FUNCTION_BLOCK FB_System_BHKW_Ablaufsteuerung
VAR_IN_OUT
	Zustand					: ST_System_BHKW_Zustand;
	Stellwert				: ST_System_BHKW_Stellwert;
	Steuerung				: ST_System_BHKW_Steuerung;
	Parameter				: ST_System_BHKW_Parameter;
END_VAR
VAR_INPUT
	Zustand_Stellventil		: ST_SVs_Zustand;
	Zustand_Pumpe			: ST_PU_Zustand;
	Zustand_BHKW			: ST_BHKW_Zustand;
END_VAR
VAR_OUTPUT
END_VAR
VAR
	Timer1					: TON;
	Timer2					: TON;
	Timer3					: TOF;
END_VAR

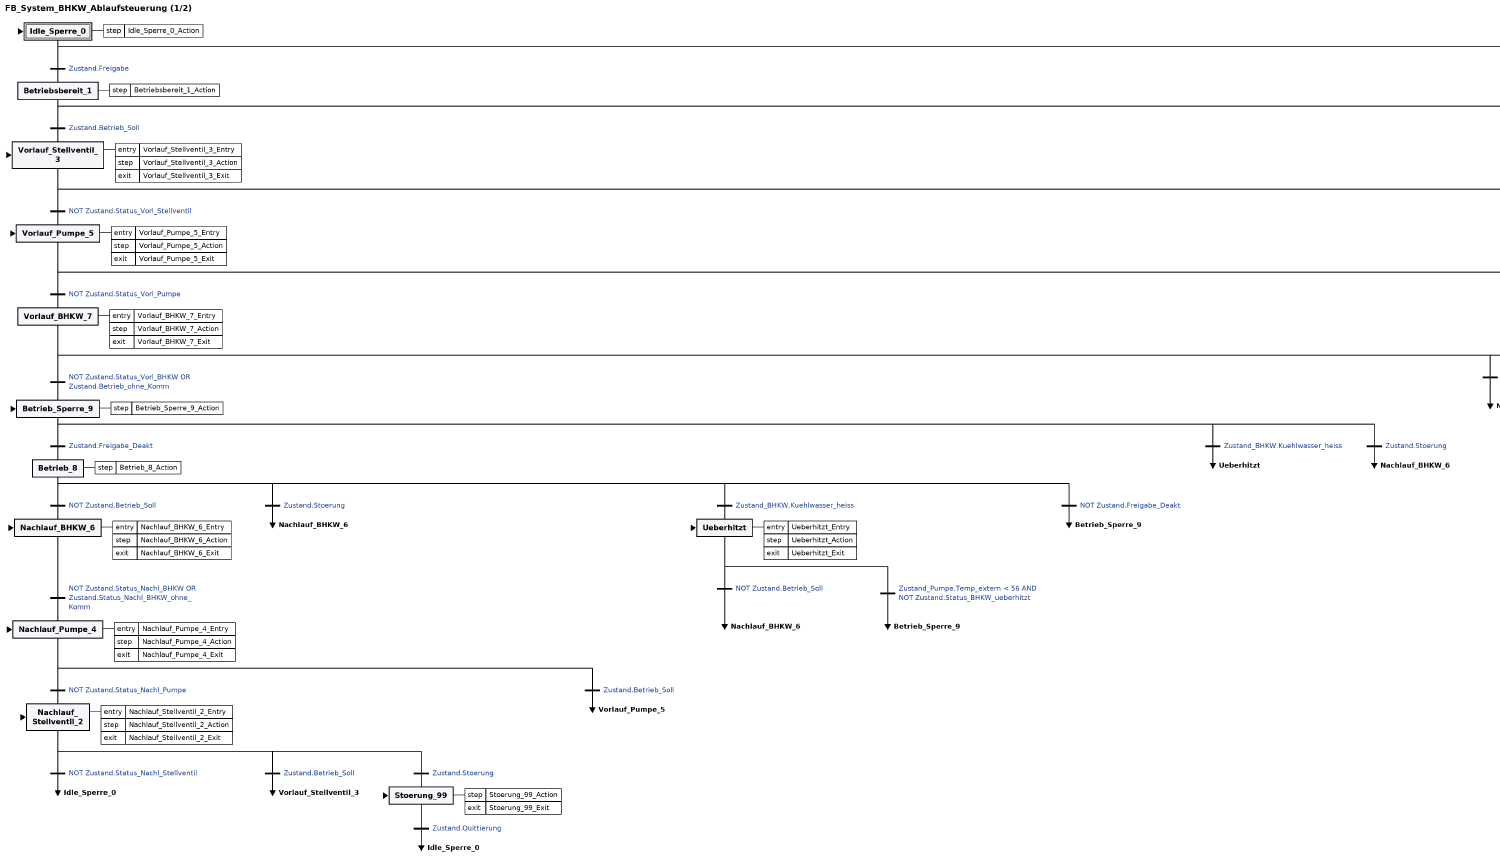
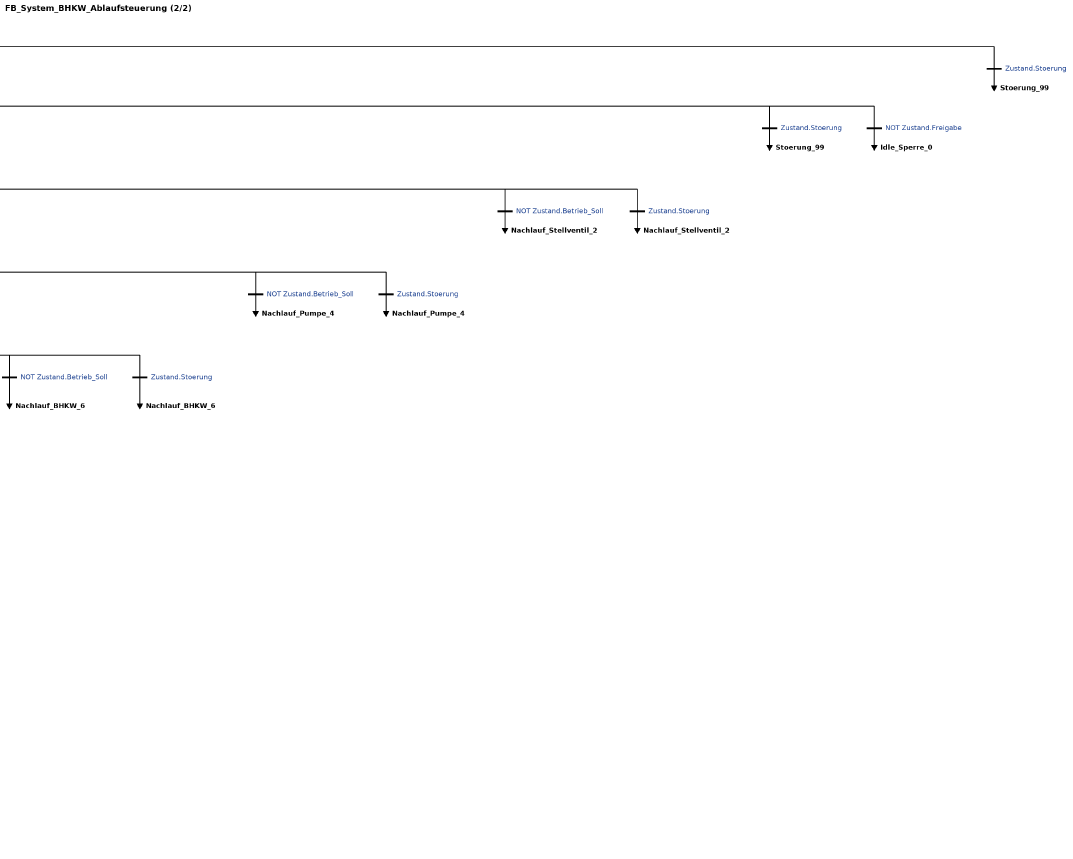
INITIAL_STEP Idle_Sperre_0:
    Idle_Sperre_0_Action(N);  // step action
END_STEP
TRANSITION FROM Idle_Sperre_0 TO Betriebsbereit_1
    := Zustand.Freigabe;
END_TRANSITION
TRANSITION FROM Idle_Sperre_0 TO Stoerung_99
    := Zustand.Stoerung;
END_TRANSITION
STEP Betriebsbereit_1:
    Betriebsbereit_1_Action(N);  // step action
END_STEP
TRANSITION FROM Betriebsbereit_1 TO Vorlauf_Stellventil_3
    := Zustand.Betrieb_Soll;
END_TRANSITION
TRANSITION FROM Betriebsbereit_1 TO Stoerung_99
    := Zustand.Stoerung;
END_TRANSITION
TRANSITION FROM Betriebsbereit_1 TO Idle_Sperre_0
    := NOT Zustand.Freigabe;
END_TRANSITION
STEP Vorlauf_Stellventil_3:
    Vorlauf_Stellventil_3_Entry(P1);  // entry action
    Vorlauf_Stellventil_3_Action(N);  // step action
    Vorlauf_Stellventil_3_Exit(P0);  // exit action
END_STEP
TRANSITION FROM Vorlauf_Stellventil_3 TO Vorlauf_Pumpe_5
    := NOT Zustand.Status_Vorl_Stellventil;
END_TRANSITION
TRANSITION FROM Vorlauf_Stellventil_3 TO Nachlauf_Stellventil_2
    := NOT Zustand.Betrieb_Soll;
END_TRANSITION
TRANSITION FROM Vorlauf_Stellventil_3 TO Nachlauf_Stellventil_2
    := Zustand.Stoerung;
END_TRANSITION
STEP Vorlauf_Pumpe_5:
    Vorlauf_Pumpe_5_Entry(P1);  // entry action
    Vorlauf_Pumpe_5_Action(N);  // step action
    Vorlauf_Pumpe_5_Exit(P0);  // exit action
END_STEP
TRANSITION FROM Vorlauf_Pumpe_5 TO Vorlauf_BHKW_7
    := NOT Zustand.Status_Vorl_Pumpe;
END_TRANSITION
TRANSITION FROM Vorlauf_Pumpe_5 TO Nachlauf_Pumpe_4
    := NOT Zustand.Betrieb_Soll;
END_TRANSITION
TRANSITION FROM Vorlauf_Pumpe_5 TO Nachlauf_Pumpe_4
    := Zustand.Stoerung;
END_TRANSITION
STEP Vorlauf_BHKW_7:
    Vorlauf_BHKW_7_Entry(P1);  // entry action
    Vorlauf_BHKW_7_Action(N);  // step action
    Vorlauf_BHKW_7_Exit(P0);  // exit action
END_STEP
TRANSITION FROM Vorlauf_BHKW_7 TO Betrieb_Sperre_9
    := NOT Zustand.Status_Vorl_BHKW OR Zustand.Betrieb_ohne_Komm;
END_TRANSITION
TRANSITION FROM Vorlauf_BHKW_7 TO Nachlauf_BHKW_6
    := NOT Zustand.Betrieb_Soll;
END_TRANSITION
TRANSITION FROM Vorlauf_BHKW_7 TO Nachlauf_BHKW_6
    := Zustand.Stoerung;
END_TRANSITION
STEP Betrieb_Sperre_9:
    Betrieb_Sperre_9_Action(N);  // step action
END_STEP
TRANSITION FROM Betrieb_Sperre_9 TO Betrieb_8
    := Zustand.Freigabe_Deakt;
END_TRANSITION
TRANSITION FROM Betrieb_Sperre_9 TO Ueberhitzt
    := Zustand_BHKW.Kuehlwasser_heiss;
END_TRANSITION
TRANSITION FROM Betrieb_Sperre_9 TO Nachlauf_BHKW_6
    := Zustand.Stoerung;
END_TRANSITION
STEP Betrieb_8:
    Betrieb_8_Action(N);  // step action
END_STEP
TRANSITION FROM Betrieb_8 TO Nachlauf_BHKW_6
    := NOT Zustand.Betrieb_Soll;
END_TRANSITION
TRANSITION FROM Betrieb_8 TO Nachlauf_BHKW_6
    := Zustand.Stoerung;
END_TRANSITION
TRANSITION FROM Betrieb_8 TO Ueberhitzt
    := Zustand_BHKW.Kuehlwasser_heiss;
END_TRANSITION
STEP Ueberhitzt:
    Ueberhitzt_Entry(P1);  // entry action
    Ueberhitzt_Action(N);  // step action
    Ueberhitzt_Exit(P0);  // exit action
END_STEP
TRANSITION FROM Ueberhitzt TO Nachlauf_BHKW_6
    := NOT Zustand.Betrieb_Soll;
END_TRANSITION
TRANSITION FROM Ueberhitzt TO Betrieb_Sperre_9
    := Zustand_Pumpe.Temp_extern < 56 AND NOT Zustand.Status_BHKW_ueberhitzt;
END_TRANSITION
TRANSITION FROM Betrieb_8 TO Betrieb_Sperre_9
    := NOT Zustand.Freigabe_Deakt;
END_TRANSITION
STEP Nachlauf_BHKW_6:
    Nachlauf_BHKW_6_Entry(P1);  // entry action
    Nachlauf_BHKW_6_Action(N);  // step action
    Nachlauf_BHKW_6_Exit(P0);  // exit action
END_STEP
TRANSITION FROM Nachlauf_BHKW_6 TO Nachlauf_Pumpe_4
    := NOT Zustand.Status_Nachl_BHKW OR Zustand.Status_Nachl_BHKW_ohne_Komm;
END_TRANSITION
STEP Nachlauf_Pumpe_4:
    Nachlauf_Pumpe_4_Entry(P1);  // entry action
    Nachlauf_Pumpe_4_Action(N);  // step action
    Nachlauf_Pumpe_4_Exit(P0);  // exit action
END_STEP
TRANSITION FROM Nachlauf_Pumpe_4 TO Nachlauf_Stellventil_2
    := NOT Zustand.Status_Nachl_Pumpe;
END_TRANSITION
TRANSITION FROM Nachlauf_Pumpe_4 TO Vorlauf_Pumpe_5
    := Zustand.Betrieb_Soll;
END_TRANSITION
STEP Nachlauf_Stellventil_2:
    Nachlauf_Stellventil_2_Entry(P1);  // entry action
    Nachlauf_Stellventil_2_Action(N);  // step action
    Nachlauf_Stellventil_2_Exit(P0);  // exit action
END_STEP
TRANSITION FROM Nachlauf_Stellventil_2 TO Idle_Sperre_0
    := NOT Zustand.Status_Nachl_Stellventil;
END_TRANSITION
TRANSITION FROM Nachlauf_Stellventil_2 TO Vorlauf_Stellventil_3
    := Zustand.Betrieb_Soll;
END_TRANSITION
TRANSITION FROM Nachlauf_Stellventil_2 TO Stoerung_99
    := Zustand.Stoerung;
END_TRANSITION
STEP Stoerung_99:
    Stoerung_99_Action(N);  // step action
    Stoerung_99_Exit(P0);  // exit action
END_STEP
TRANSITION FROM Stoerung_99 TO Idle_Sperre_0
    := Zustand.Quittierung;
END_TRANSITION

ACTION Betrieb_8_Action:
(* Stellwert setzen *)
Stellwert.Anford_Stellventil		:= TRUE;
Stellwert.Anford_Pumpe		:= TRUE;
Stellwert.Anford_BHKW			:= TRUE;

(* Zustand setzen *)
Zustand.Status				:= E_System_BHKW_Zustand_Status_Betrieb;
END_ACTION

ACTION Betrieb_Sperre_9_Action:
(* Stellwert setzen *)
Stellwert.Anford_Stellventil		:= TRUE;
Stellwert.Anford_Pumpe		:= TRUE;
Stellwert.Anford_BHKW			:= TRUE;

(* Zustand setzen *)
Zustand.Status				:= E_System_BHKW_Zustand_Status_Betrieb_Sperre;
END_ACTION

ACTION Betriebsbereit_1_Action:
(* Stellwert setzen *)
Stellwert.Anford_Stellventil	:= FALSE;
Stellwert.Anford_Pumpe	:= FALSE;
Stellwert.Anford_BHKW		:= FALSE;

(* Zustand setzen *)
Zustand.Status			:= E_System_BHKW_Zustand_Status_Betriebsbereit;
END_ACTION

ACTION Idle_Sperre_0_Action:
(* Stellwert setzen *)
Stellwert.Anford_Stellventil	:= FALSE;
Stellwert.Anford_Pumpe	:= FALSE;
Stellwert.Anford_BHKW		:= FALSE;

(* Zustand setzen *)
Zustand.Status			:= E_System_BHKW_Zustand_Status_Idle_Sperre;
Zustand.Betrieb_ohne_Komm	:= FALSE;


(* Quittierungszustand auf False setzen, damit das System bei einer erneuten Störung nicht direkt wieder angeschaltet wird *)
Steuerung.Quittierung	:= FALSE;
END_ACTION

ACTION Nachlauf_BHKW_6_Action:
(* Stellwert setzen *)
Stellwert.Anford_Stellventil		:= TRUE;
Stellwert.Anford_Pumpe		:= TRUE;
Stellwert.Anford_BHKW			:= FALSE;

(* Zustand setzen *)
Zustand.Status				:= E_System_BHKW_Zustand_Status_Nachl_BHKW;
Zustand_BHKW.Status_Nachl;
Zustand.Status_Nachl_BHKW	:= Zustand_BHKW.Betrieb OR Zustand_BHKW.Status_Nachl;


(* falls es keine Rückmeldung vom BHKW-Kommunikationsmodul gibt, geht der Nachlauf dennoch weiter *)
Timer2(	IN := Zustand.Status_Nachl_BHKW,
		PT := Parameter.Zeit_Nachl,
		Q => Zustand.Status_Nachl_BHKW_ohne_Komm
);
Zustand.Status_Nachl_BHKW_ohne_Komm := NOT Zustand.Status_Nachl_BHKW_ohne_Komm;
END_ACTION

ACTION Nachlauf_BHKW_6_Entry:
Zustand.Status_Nachl_BHKW			:= TRUE;
Zustand.Status_Nachl_BHKW_ohne_Komm := TRUE;
END_ACTION

ACTION Nachlauf_BHKW_6_Exit:
Zustand.Status_Nachl_BHKW			:= FALSE;
Zustand.Status_Nachl_BHKW_ohne_Komm := FALSE;
END_ACTION

ACTION Nachlauf_Pumpe_4_Action:
(* Stellwert setzen *)
Stellwert.Anford_Stellventil		:= TRUE;
Stellwert.Anford_Pumpe				:= FALSE;
Stellwert.Anford_BHKW				:= FALSE;

(* Zustand setzen *)
Zustand.Status				:= E_System_BHKW_Zustand_Status_Nachl_Pumpe;
Zustand.Status_Nachl_Pumpe	:= Zustand_Pumpe.Betrieb OR Zustand_Pumpe.Status_Nachl;
END_ACTION

ACTION Nachlauf_Pumpe_4_Entry:
Zustand.Status_Nachl_Pumpe	:= TRUE;
END_ACTION

ACTION Nachlauf_Pumpe_4_Exit:
Zustand.Status_Nachl_Pumpe	:= FALSE;
END_ACTION

ACTION Nachlauf_Stellventil_2_Action:
(* Stellwert setzen *)
Stellwert.Anford_Stellventil		:= FALSE;
Stellwert.Anford_Pumpe		:= FALSE;
Stellwert.Anford_BHKW			:= FALSE;

(* Zustand setzen *)
Zustand.Status				:= E_System_BHKW_Zustand_Status_Nachl_Stellventil;
Zustand.Status_Nachl_Stellventil	:= Zustand_Stellventil.Stellung OR Zustand_Stellventil.Stellungwechsel10;
END_ACTION

ACTION Nachlauf_Stellventil_2_Entry:
Zustand.Status_Nachl_Stellventil	:= TRUE;
END_ACTION

ACTION Nachlauf_Stellventil_2_Exit:
Zustand.Status_Nachl_Stellventil	:= FALSE;
END_ACTION

ACTION Stoerung_99_Action:
(* Stellwert setzen *)
Stellwert.Anford_Stellventil	:= FALSE;
Stellwert.Anford_Pumpe	:= FALSE;
Stellwert.Anford_BHKW		:= FALSE;

(* Zustand setzen *)
Zustand.Stoerung			:= TRUE;
Zustand.Status			:= E_System_BHKW_Zustand_Status_Stoerung;
END_ACTION

ACTION Stoerung_99_Exit:
Zustand.Stoerung	:= FALSE;
END_ACTION

ACTION Ueberhitzt_Action:
(* Stellwert setzen *)
Stellwert.Anford_Stellventil	:= TRUE;
Stellwert.Anford_Pumpe			:= TRUE;
Stellwert.Anford_BHKW			:= FALSE;

(* Zustand setzen *)
Zustand.Status				:= E_System_BHKW_Zustand_Status_Ueberhitzt;

(* Mindestens eine halbe Stunde abkühlen *)
Timer3( IN := Zustand_BHKW.Kuehlwasser_heiss,
		PT := T#30M
);

Zustand.Status_BHKW_ueberhitzt := Timer3.Q;
END_ACTION

ACTION Ueberhitzt_Entry:
Zustand.Status_BHKW_ueberhitzt := TRUE;
(* Reset Timer *)
Timer3(IN := FALSE);
END_ACTION

ACTION Ueberhitzt_Exit:
Zustand.Status_BHKW_ueberhitzt := FALSE;
(* Reset Timer *)
Timer3(IN := FALSE);
END_ACTION

ACTION Vorlauf_BHKW_7_Action:
(* Stellwert setzen *)
Stellwert.Anford_Stellventil		:= TRUE;
Stellwert.Anford_Pumpe		:= TRUE;
Stellwert.Anford_BHKW			:= TRUE;

(* Zustand setzen *)
Zustand.Status				:= E_System_BHKW_Zustand_Status_Vorl_BHKW;
Zustand.Status_Vorl_BHKW		:= NOT(Zustand_BHKW.Betrieb AND NOT Zustand_BHKW.Status_Vorl);


(* falls keine Rückmeldung vom BHKW-Kommunikationsmodul kommt, wird der Zustand dennoch auf Betrieb gesetzt *)
Timer1(	IN := Zustand.Status_Vorl_BHKW,
		PT := Parameter.Zeit_Vorl,
		Q => Zustand.Betrieb_ohne_Komm
);
END_ACTION

ACTION Vorlauf_BHKW_7_Entry:
Zustand.Status_Vorl_BHKW		:= TRUE;
END_ACTION

ACTION Vorlauf_BHKW_7_Exit:
Zustand.Status_Vorl_BHKW		:= FALSE;
END_ACTION

ACTION Vorlauf_Pumpe_5_Action:
(* Stellwert setzen *)
Stellwert.Anford_Stellventil		:= TRUE;
Stellwert.Anford_Pumpe		:= TRUE;
Stellwert.Anford_BHKW			:= FALSE;

(* Zustand setzen *)
Zustand.Status				:= E_System_BHKW_Zustand_Status_Vorl_Pumpe;
Zustand.Status_Vorl_Pumpe	:= NOT(Zustand_Pumpe.Betrieb AND NOT Zustand_Pumpe.Status_Vorl);
END_ACTION

ACTION Vorlauf_Pumpe_5_Entry:
Zustand.Status_Vorl_Pumpe	:= TRUE;
END_ACTION

ACTION Vorlauf_Pumpe_5_Exit:
Zustand.Status_Vorl_Pumpe	:= FALSE;
END_ACTION

ACTION Vorlauf_Stellventil_3_Action:
(* Stellwert setzen *)
Stellwert.Anford_Stellventil		:= TRUE;
Stellwert.Anford_Pumpe		:= FALSE;
Stellwert.Anford_BHKW			:= FALSE;

(* Zustand setzen *)
Zustand.Status				:= E_System_BHKW_Zustand_Status_Vorl_Stellventil;
Zustand.Status_Vorl_Stellventil	:= NOT(Zustand_Stellventil.Stellung AND NOT Zustand_Stellventil.Stellungwechsel01);
END_ACTION

ACTION Vorlauf_Stellventil_3_Entry:
Zustand.Status_Vorl_Stellventil	:= TRUE;
END_ACTION

ACTION Vorlauf_Stellventil_3_Exit:
Zustand.Status_Vorl_Stellventil	:= FALSE;
END_ACTION

END_FUNCTION_BLOCK

(* stored: Version 1.1.0.1, ProductVersion 3.1.4024.9
   POU FB_System_BHKW_Ablaufsteuerung: Id {0d992d6a-17ae-4c9a-9175-b7ad9042449e}, SpecialFunc None
   Action Betrieb_8_Action: Id {f6ff5d91-81a1-47e3-9b11-3a1fb931e0b7}
   Action Betrieb_Sperre_9_Action: Id {15e2f310-2d34-48a0-be6c-a857e905243b}
   Action Betriebsbereit_1_Action: Id {ddbbdb63-a1bf-48ca-b983-522025ac87f9}
   Action Idle_Sperre_0_Action: Id {874ad14d-8c51-4b06-9382-66e85d0b7f8f}
   Action Nachlauf_BHKW_6_Action: Id {0863fcf4-35d7-47f1-b154-494e918f2f29}
   Action Nachlauf_BHKW_6_Entry: Id {e06191bc-b68e-47be-86a0-865ce1eb0598}
   Action Nachlauf_BHKW_6_Exit: Id {6a833044-395d-4cba-b5ea-130f298bbcde}
   Action Nachlauf_Pumpe_4_Action: Id {7b5ade18-f868-41ae-811f-a0bd93b73cdf}
   Action Nachlauf_Pumpe_4_Entry: Id {b3d9f5a9-6865-43fe-a484-0dc60f2e6734}
   Action Nachlauf_Pumpe_4_Exit: Id {3c158ca3-3d19-4321-94cb-984e751f7e1d}
   Action Nachlauf_Stellventil_2_Action: Id {94a87d77-1b30-4ac1-981c-58a93acf7bb9}
   Action Nachlauf_Stellventil_2_Entry: Id {238bb23c-faf7-475b-9491-c9652e577398}
   Action Nachlauf_Stellventil_2_Exit: Id {304f461b-f8bd-45ee-a08c-4db7f0156585}
   Action Stoerung_99_Action: Id {0864472b-7aef-4809-bc31-21ebc0716359}
   Action Stoerung_99_Exit: Id {629dfc7c-53d0-41a7-b8d9-8d9f80187169}
   Action Ueberhitzt_Action: Id {b539ce05-b469-4d97-986e-41f78b5b1d4e}
   Action Ueberhitzt_Entry: Id {15f67544-2a54-4a86-a1b2-84b25abc8819}
   Action Ueberhitzt_Exit: Id {38aee387-8389-4fb7-ae81-6c829f938e37}
   Action Vorlauf_BHKW_7_Action: Id {4aa35037-d346-45af-bea4-b486b62d2d2f}
   Action Vorlauf_BHKW_7_Entry: Id {38426a22-1167-4f7d-8b31-f7ec2b33fdb0}
   Action Vorlauf_BHKW_7_Exit: Id {bc03f656-9483-4522-81e5-bb98ef89ac5a}
   Action Vorlauf_Pumpe_5_Action: Id {696fa86c-d0f6-44b7-afdd-ae7c6a00b492}
   Action Vorlauf_Pumpe_5_Entry: Id {6e1af50a-8098-48f9-bc17-2b281b4aec11}
   Action Vorlauf_Pumpe_5_Exit: Id {4cb717b8-bd61-4aff-bb18-5e653863f0f9}
   Action Vorlauf_Stellventil_3_Action: Id {fdd78b54-fec3-4406-afbf-36a594508323}
   Action Vorlauf_Stellventil_3_Entry: Id {98a8c424-9de5-4ffb-8ebf-06038bb8211c}
   Action Vorlauf_Stellventil_3_Exit: Id {01bc1713-6f6d-4de2-b3c1-2956be503106} *)
